// SIMATIC S7-200 project (STEP 7-Micro/WIN), CPU 224 CN REL 02.01

SYMBOL_TABLE 用户定义1
缺料故障             M11.3
急停故障             M11.2
立箱不成功故障          M11.1
折盖回              T99
上升               Q1.0
下降               Q1.1
主机零位脉冲           M4.1
系统运行             M4.0
主机零位接近           I0.1
启动               I1.1
停止               I1.2
复位               I2.5
缺料光电             I2.2
红灯               Q0.2
绿灯               Q0.3
黄灯               Q0.5
主1速              Q0.4
主2速              Q0.6
主3速              Q0.7
吸箱真空             Q2.0
吸箱气缸             Q2.1
抹箱               Q2.3
折盖               Q2.4
固箱               Q2.5
上夹               Q2.6
下放               Q2.7
固箱真空             Q3.1
左推               Q3.2
右推               Q3.3
屏启动              V10.0
屏停止              V10.1
停箱脉冲光电           I2.7
满箱报警             M13.3
满箱光电             I1.0
END_SYMBOL_TABLE

ORGANIZATION_BLOCK 主程序:OB1
TITLE=程序注释
BEGIN
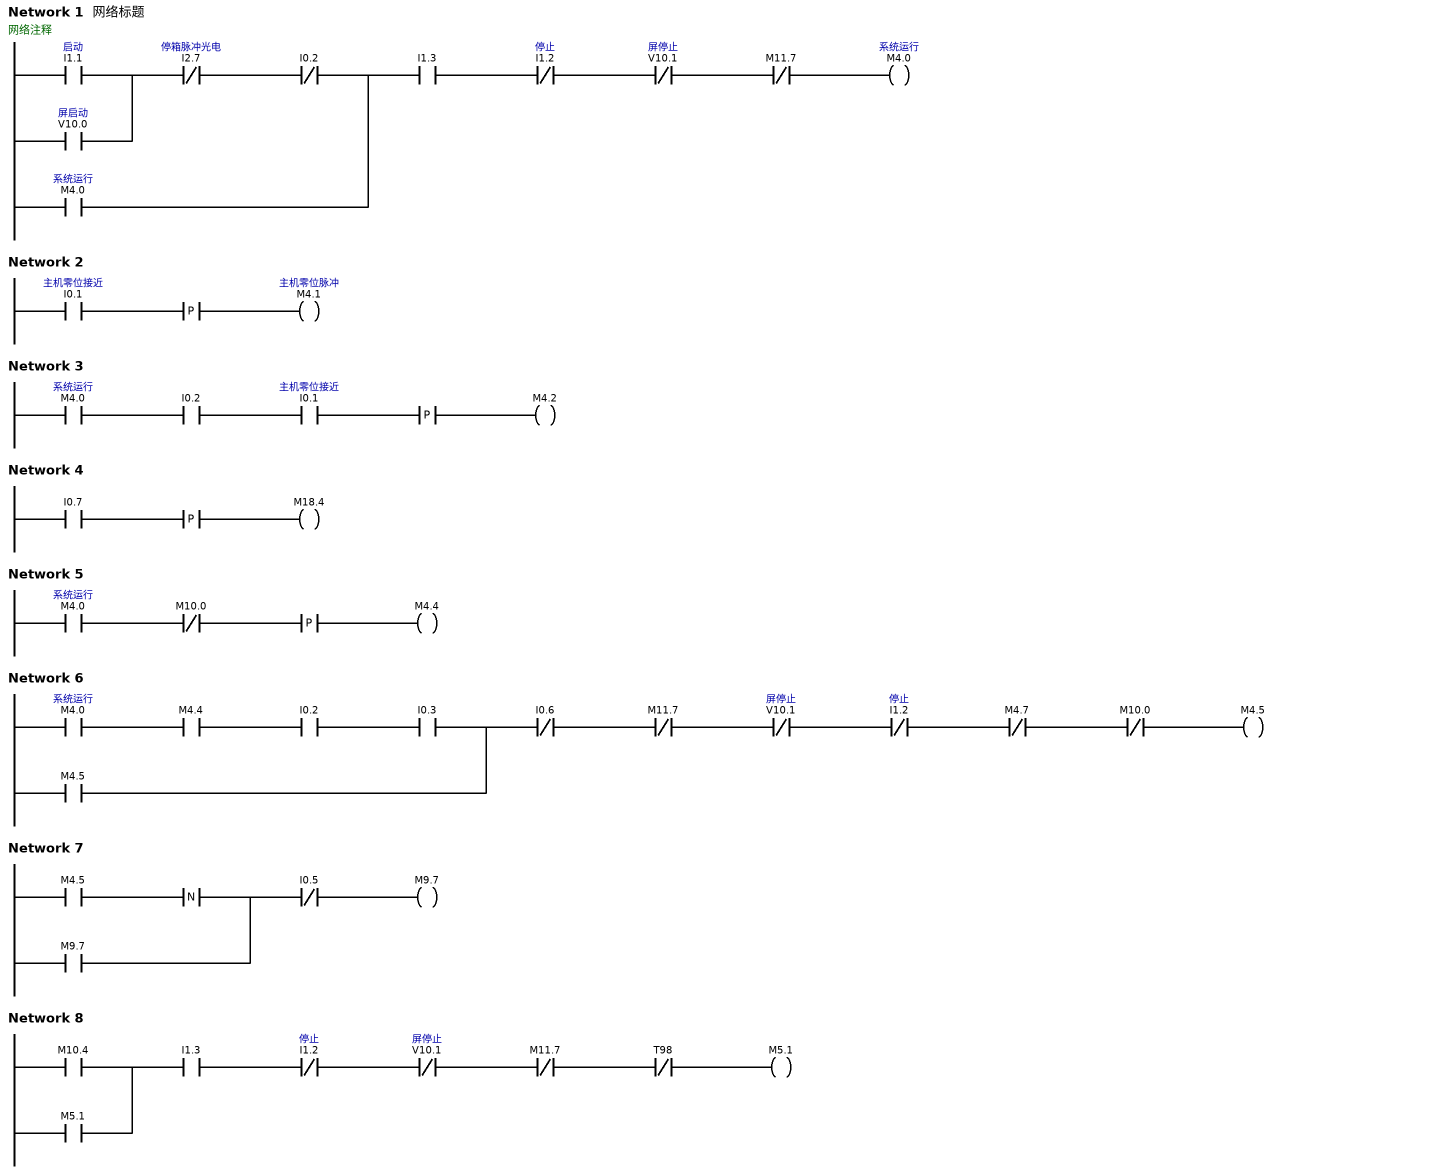
Network 1 // 网络标题
// 网络注释
LD     启动:I1.1
O      屏启动:V10.0
AN     停箱脉冲光电:I2.7
AN     I0.2
O      系统运行:M4.0
A      I1.3
AN     停止:I1.2
AN     屏停止:V10.1
AN     M11.7
=      系统运行:M4.0
Network 2
LD     主机零位接近:I0.1
EU
=      主机零位脉冲:M4.1
Network 3
LD     系统运行:M4.0
A      I0.2
A      主机零位接近:I0.1
EU
=      M4.2
Network 4
LD     I0.7
EU
=      M18.4
Network 5
LD     系统运行:M4.0
AN     M10.0
EU
=      M4.4
Network 6
LD     系统运行:M4.0
A      M4.4
A      I0.2
A      I0.3
O      M4.5
AN     I0.6
AN     M11.7
AN     屏停止:V10.1
AN     停止:I1.2
AN     M4.7
AN     M10.0
=      M4.5
Network 7
LD     M4.5
ED
O      M9.7
AN     I0.5
=      M9.7
Network 8
LD     M10.4
O      M5.1
A      I1.3
AN     停止:I1.2
AN     屏停止:V10.1
AN     M11.7
AN     T98
=      M5.1
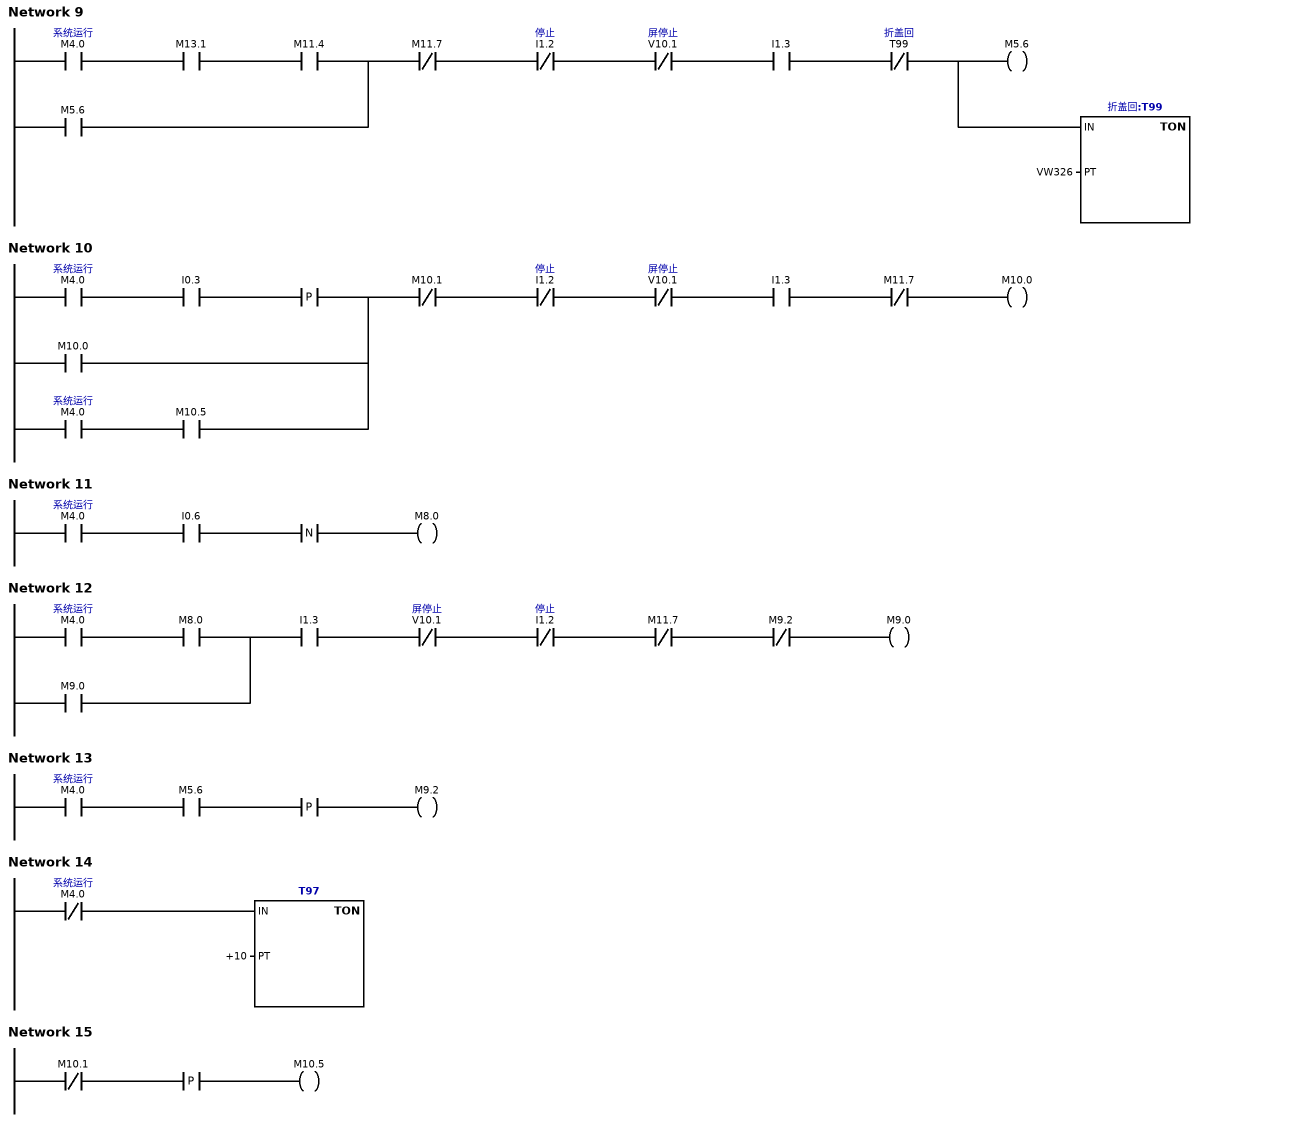
Network 9
LD     系统运行:M4.0
A      M13.1
A      M11.4
O      M5.6
AN     M11.7
AN     停止:I1.2
AN     屏停止:V10.1
A      I1.3
AN     折盖回:T99
=      M5.6
TON    折盖回:T99, VW326
Network 10
LD     系统运行:M4.0
A      I0.3
EU
O      M10.0
LD     系统运行:M4.0
A      M10.5
OLD
AN     M10.1
AN     停止:I1.2
AN     屏停止:V10.1
A      I1.3
AN     M11.7
=      M10.0
Network 11
LD     系统运行:M4.0
A      I0.6
ED
=      M8.0
Network 12
LD     系统运行:M4.0
A      M8.0
O      M9.0
A      I1.3
AN     屏停止:V10.1
AN     停止:I1.2
AN     M11.7
AN     M9.2
=      M9.0
Network 13
LD     系统运行:M4.0
A      M5.6
EU
=      M9.2
Network 14
LDN    系统运行:M4.0
TON    T97, +10
Network 15
LDN    M10.1
EU
=      M10.5
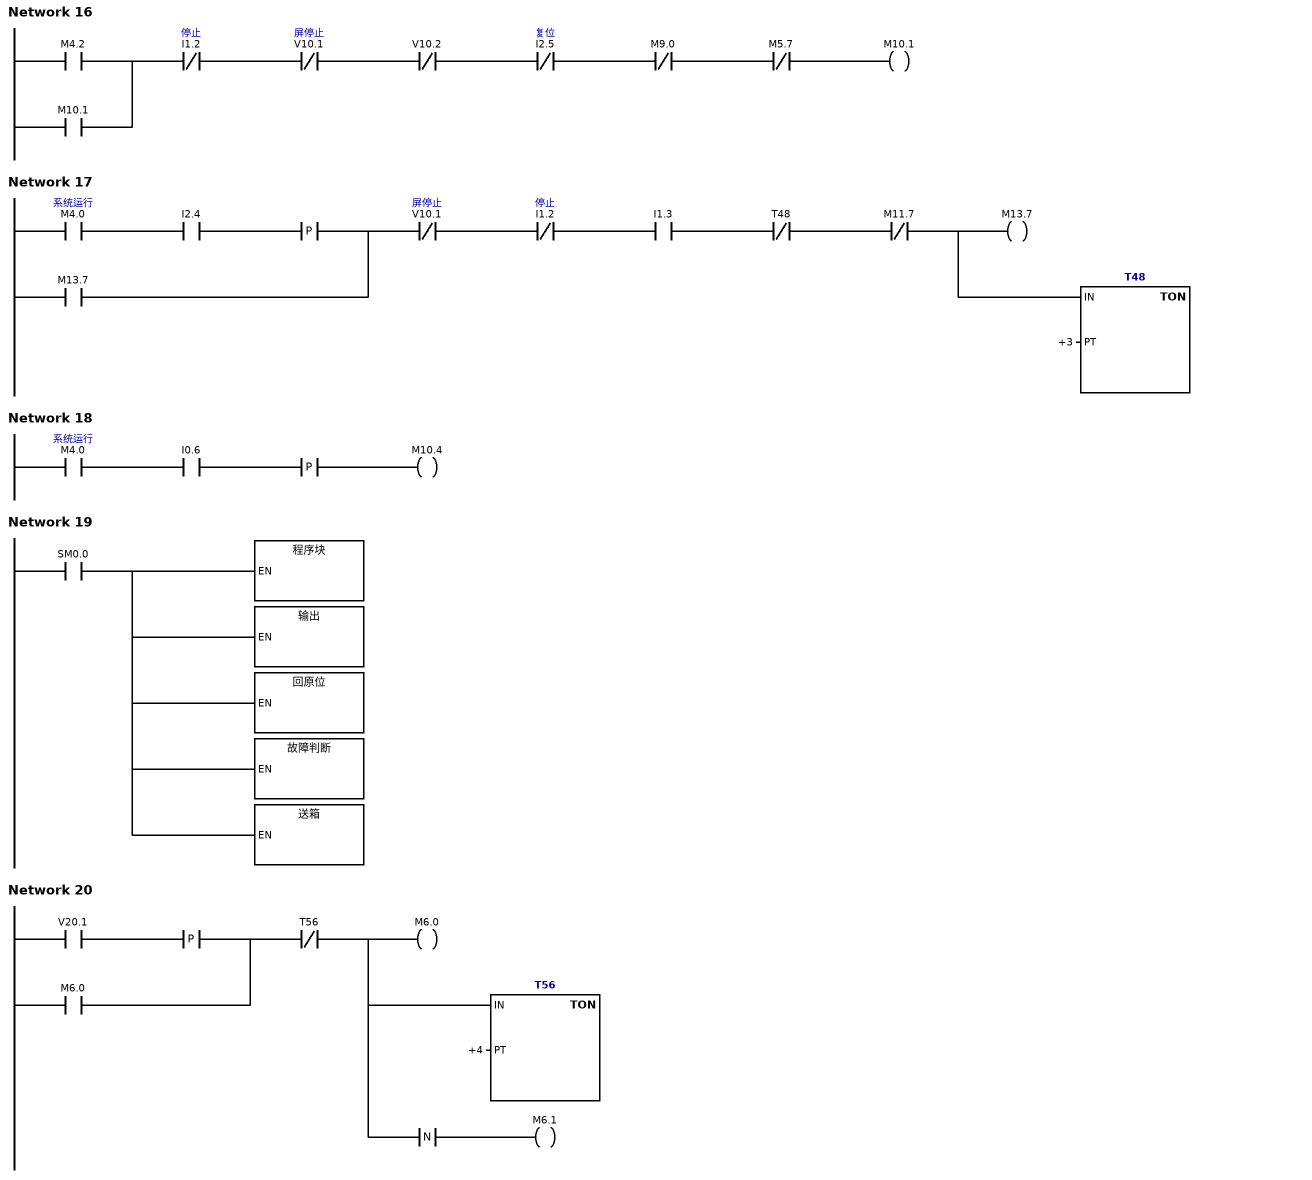
Network 16
LD     M4.2
O      M10.1
AN     停止:I1.2
AN     屏停止:V10.1
AN     V10.2
AN     复位:I2.5
AN     M9.0
AN     M5.7
=      M10.1
Network 17
LD     系统运行:M4.0
A      I2.4
EU
O      M13.7
AN     屏停止:V10.1
AN     停止:I1.2
A      I1.3
AN     T48
AN     M11.7
=      M13.7
TON    T48, +3
Network 18
LD     系统运行:M4.0
A      I0.6
EU
=      M10.4
Network 19
LD     SM0.0
CALL   程序块:SBR0
CALL   输出:SBR1
CALL   回原位:SBR4
CALL   故障判断:SBR3
CALL   送箱:SBR2
Network 20
LD     V20.1
EU
O      M6.0
AN     T56
=      M6.0
TON    T56, +4
ED
=      M6.1
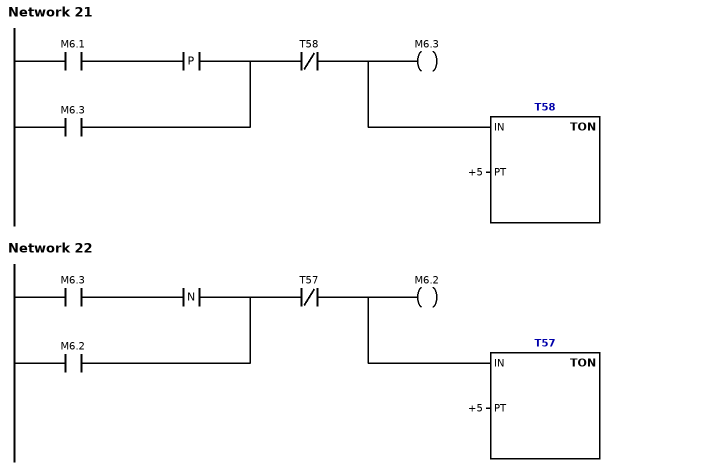
Network 21
LD     M6.1
EU
O      M6.3
AN     T58
=      M6.3
TON    T58, +5
Network 22
LD     M6.3
ED
O      M6.2
AN     T57
=      M6.2
TON    T57, +5
END_ORGANIZATION_BLOCK

SUBROUTINE_BLOCK 程序块:SBR0
TITLE=子程序注释
BEGIN
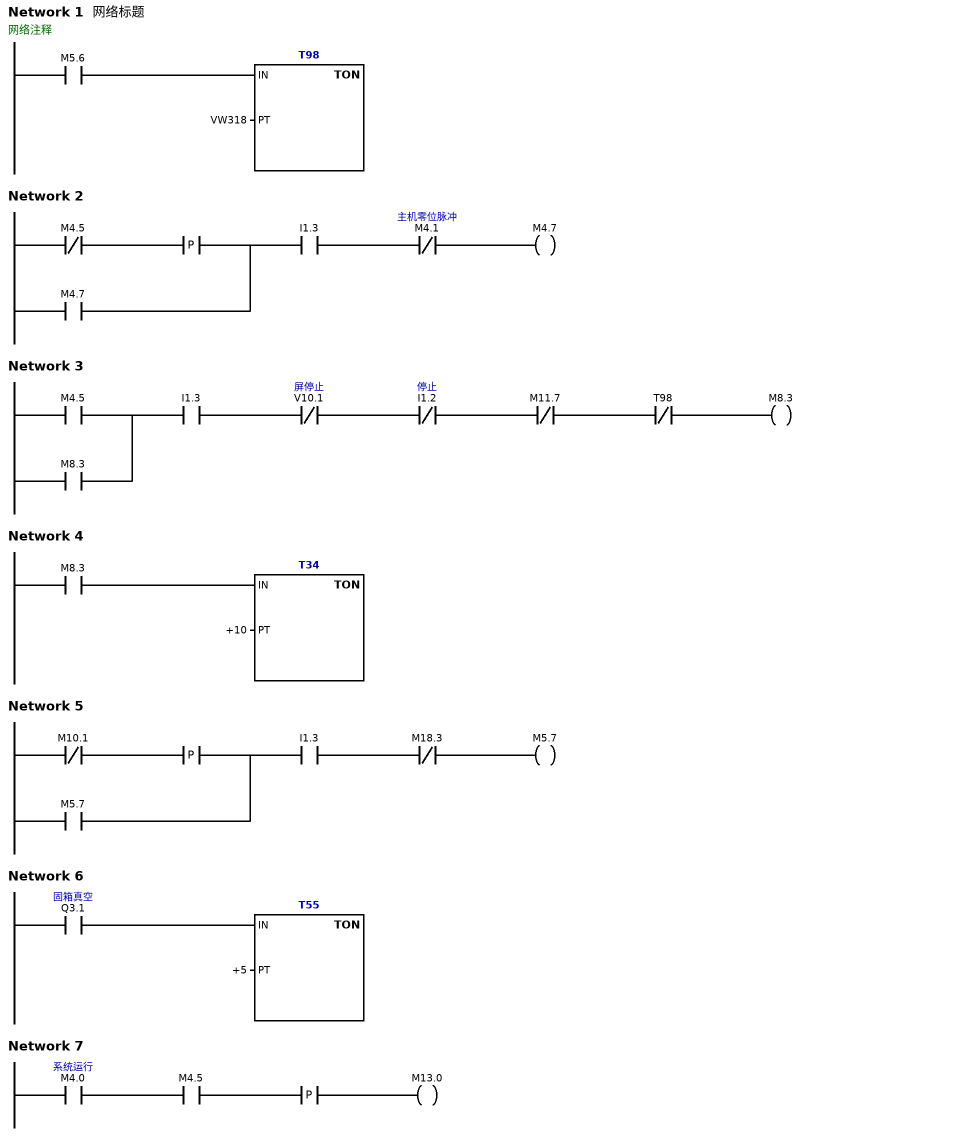
Network 1 // 网络标题
// 网络注释
LD     M5.6
TON    T98, VW318
Network 2
LDN    M4.5
EU
O      M4.7
A      I1.3
AN     主机零位脉冲:M4.1
=      M4.7
Network 3
LD     M4.5
O      M8.3
A      I1.3
AN     屏停止:V10.1
AN     停止:I1.2
AN     M11.7
AN     T98
=      M8.3
Network 4
LD     M8.3
TON    T34, +10
Network 5
LDN    M10.1
EU
O      M5.7
A      I1.3
AN     M18.3
=      M5.7
Network 6
LD     固箱真空:Q3.1
TON    T55, +5
Network 7
LD     系统运行:M4.0
A      M4.5
EU
=      M13.0
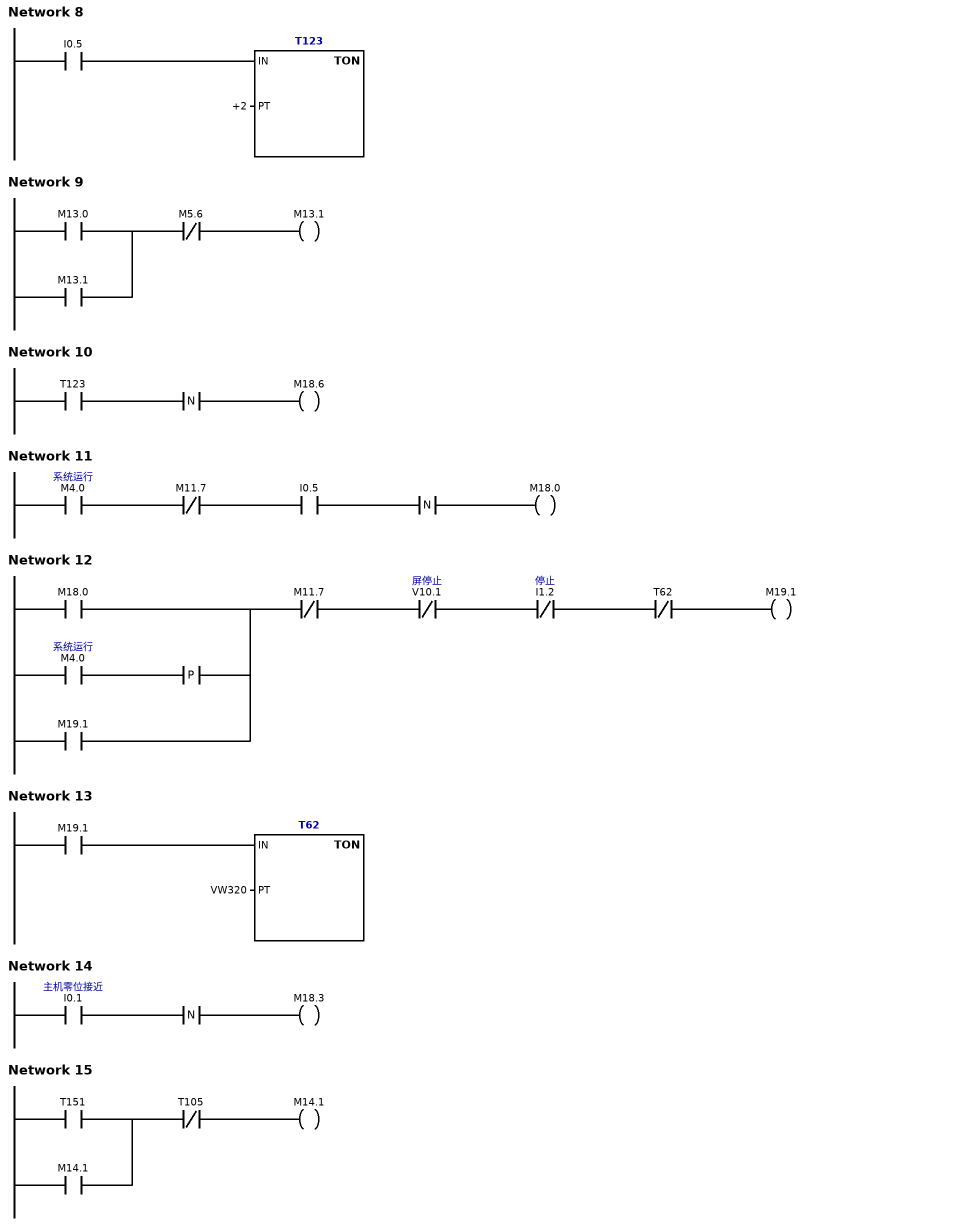
Network 8
LD     I0.5
TON    T123, +2
Network 9
LD     M13.0
O      M13.1
AN     M5.6
=      M13.1
Network 10
LD     T123
ED
=      M18.6
Network 11
LD     系统运行:M4.0
AN     M11.7
A      I0.5
ED
=      M18.0
Network 12
LD     M18.0
LD     系统运行:M4.0
EU
OLD
O      M19.1
AN     M11.7
AN     屏停止:V10.1
AN     停止:I1.2
AN     T62
=      M19.1
Network 13
LD     M19.1
TON    T62, VW320
Network 14
LD     主机零位接近:I0.1
ED
=      M18.3
Network 15
LD     T151
O      M14.1
AN     T105
=      M14.1
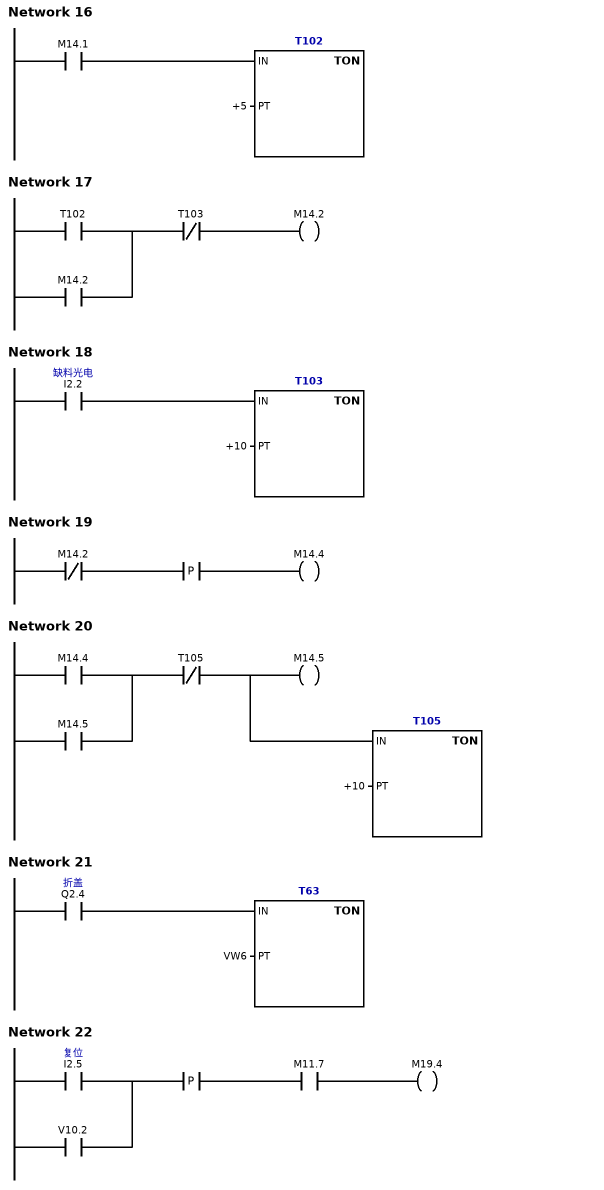
Network 16
LD     M14.1
TON    T102, +5
Network 17
LD     T102
O      M14.2
AN     T103
=      M14.2
Network 18
LD     缺料光电:I2.2
TON    T103, +10
Network 19
LDN    M14.2
EU
=      M14.4
Network 20
LD     M14.4
O      M14.5
AN     T105
=      M14.5
TON    T105, +10
Network 21
LD     折盖:Q2.4
TON    T63, VW6
Network 22
LD     复位:I2.5
O      V10.2
EU
A      M11.7
=      M19.4
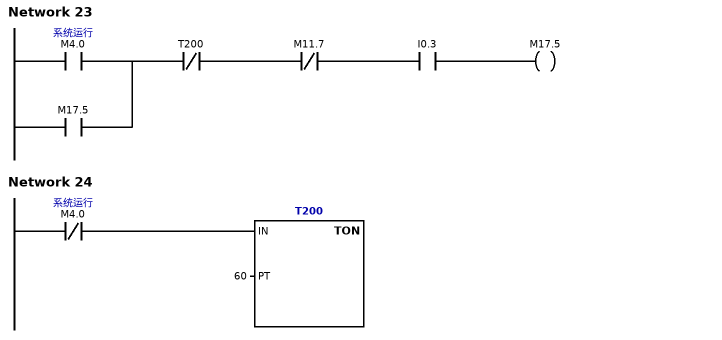
Network 23
LD     系统运行:M4.0
O      M17.5
AN     T200
AN     M11.7
A      I0.3
=      M17.5
Network 24
LDN    系统运行:M4.0
TON    T200, 60
END_SUBROUTINE_BLOCK

SUBROUTINE_BLOCK 输出:SBR1
TITLE=子程序注释
BEGIN
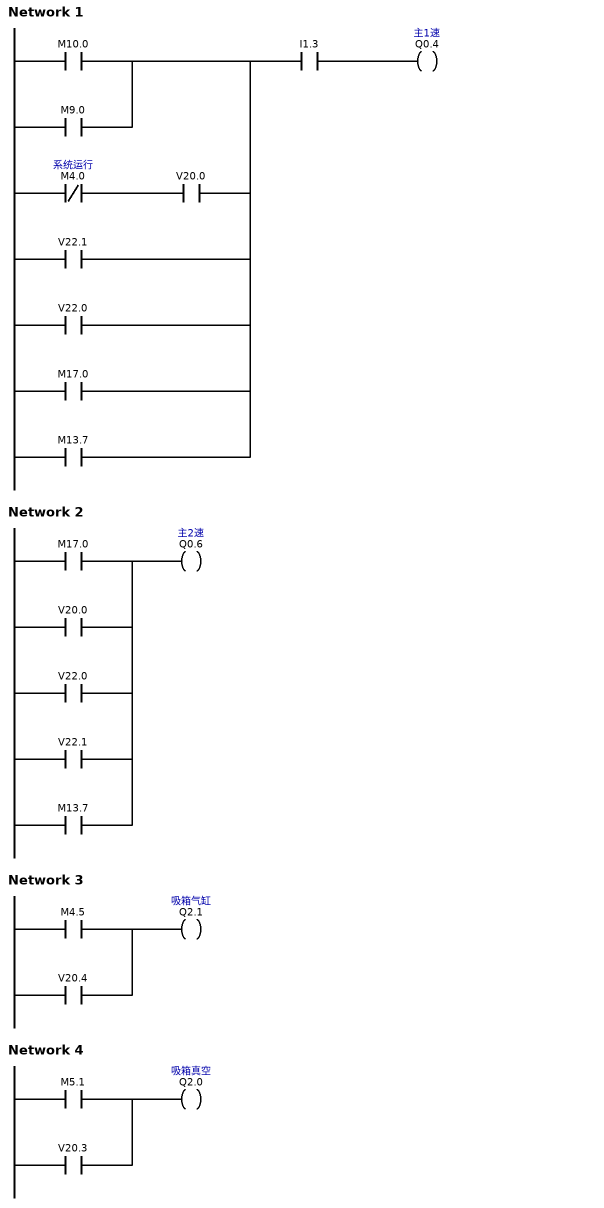
Network 1
LD     M10.0
O      M9.0
LDN    系统运行:M4.0
A      V20.0
OLD
O      V22.1
O      V22.0
O      M17.0
O      M13.7
A      I1.3
=      主1速:Q0.4
Network 2
LD     M17.0
O      V20.0
O      V22.0
O      V22.1
O      M13.7
=      主2速:Q0.6
Network 3
LD     M4.5
O      V20.4
=      吸箱气缸:Q2.1
Network 4
LD     M5.1
O      V20.3
=      吸箱真空:Q2.0
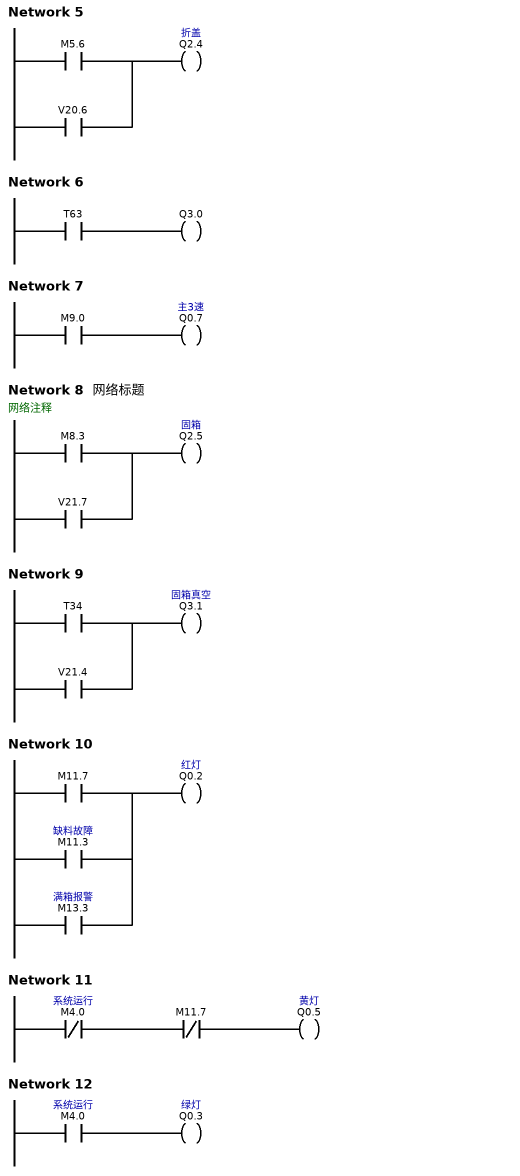
Network 5
LD     M5.6
O      V20.6
=      折盖:Q2.4
Network 6
LD     T63
=      Q3.0
Network 7
LD     M9.0
=      主3速:Q0.7
Network 8 // 网络标题
// 网络注释
LD     M8.3
O      V21.7
=      固箱:Q2.5
Network 9
LD     T34
O      V21.4
=      固箱真空:Q3.1
Network 10
LD     M11.7
O      缺料故障:M11.3
O      满箱报警:M13.3
=      红灯:Q0.2
Network 11
LDN    系统运行:M4.0
AN     M11.7
=      黄灯:Q0.5
Network 12
LD     系统运行:M4.0
=      绿灯:Q0.3
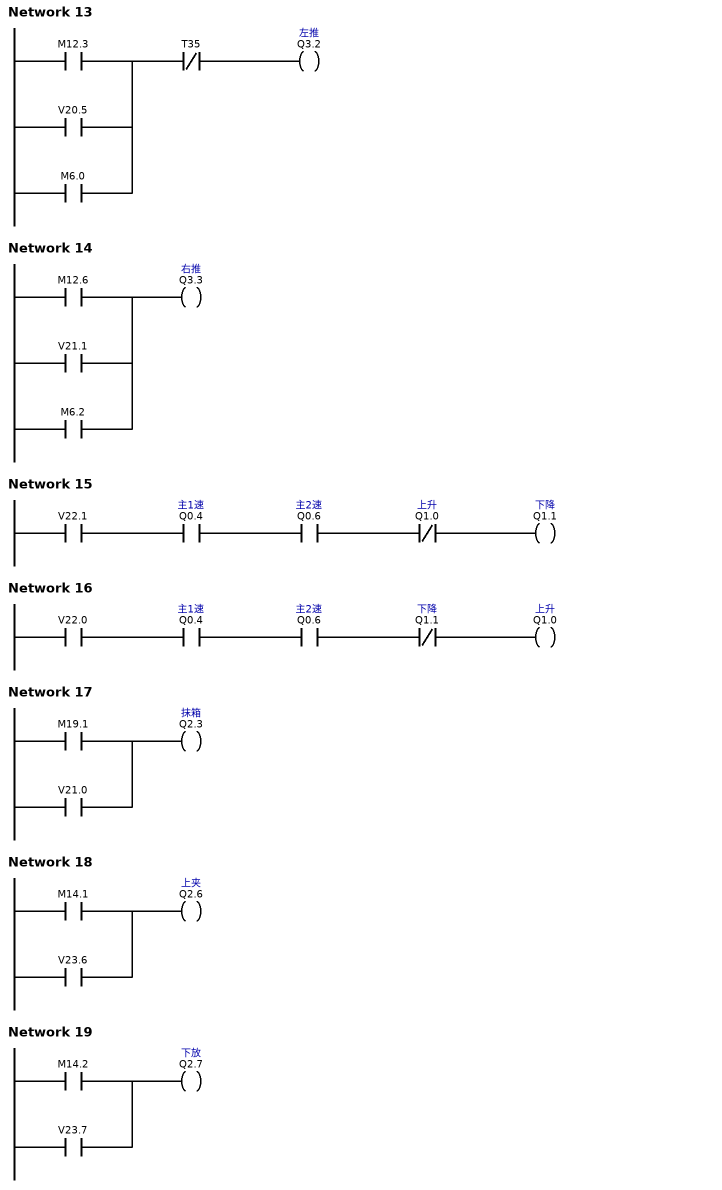
Network 13
LD     M12.3
O      V20.5
O      M6.0
AN     T35
=      左推:Q3.2
Network 14
LD     M12.6
O      V21.1
O      M6.2
=      右推:Q3.3
Network 15
LD     V22.1
A      主1速:Q0.4
A      主2速:Q0.6
AN     上升:Q1.0
=      下降:Q1.1
Network 16
LD     V22.0
A      主1速:Q0.4
A      主2速:Q0.6
AN     下降:Q1.1
=      上升:Q1.0
Network 17
LD     M19.1
O      V21.0
=      抹箱:Q2.3
Network 18
LD     M14.1
O      V23.6
=      上夹:Q2.6
Network 19
LD     M14.2
O      V23.7
=      下放:Q2.7
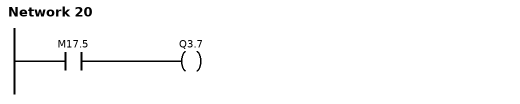
Network 20
LD     M17.5
=      Q3.7
END_SUBROUTINE_BLOCK

SUBROUTINE_BLOCK 送箱:SBR2
TITLE=子程序注释
BEGIN
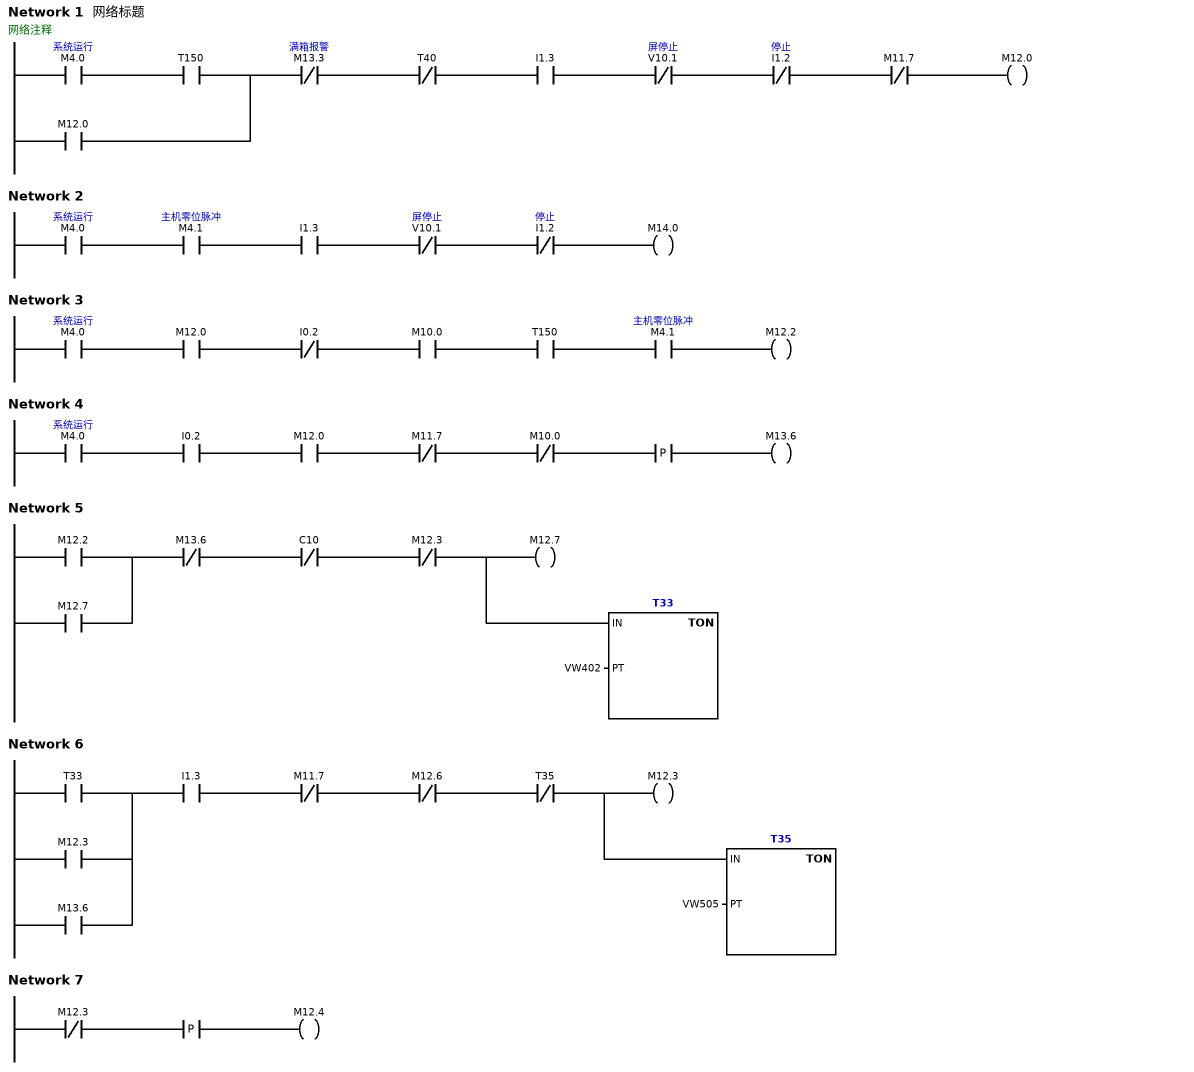
Network 1 // 网络标题
// 网络注释
LD     系统运行:M4.0
A      T150
O      M12.0
AN     满箱报警:M13.3
AN     T40
A      I1.3
AN     屏停止:V10.1
AN     停止:I1.2
AN     M11.7
=      M12.0
Network 2
LD     系统运行:M4.0
A      主机零位脉冲:M4.1
A      I1.3
AN     屏停止:V10.1
AN     停止:I1.2
=      M14.0
Network 3
LD     系统运行:M4.0
A      M12.0
AN     I0.2
A      M10.0
A      T150
A      主机零位脉冲:M4.1
=      M12.2
Network 4
LD     系统运行:M4.0
A      I0.2
A      M12.0
AN     M11.7
AN     M10.0
EU
=      M13.6
Network 5
LD     M12.2
O      M12.7
AN     M13.6
AN     C10
AN     M12.3
=      M12.7
TON    T33, VW402
Network 6
LD     T33
O      M12.3
O      M13.6
A      I1.3
AN     M11.7
AN     M12.6
AN     T35
=      M12.3
TON    T35, VW505
Network 7
LDN    M12.3
EU
=      M12.4
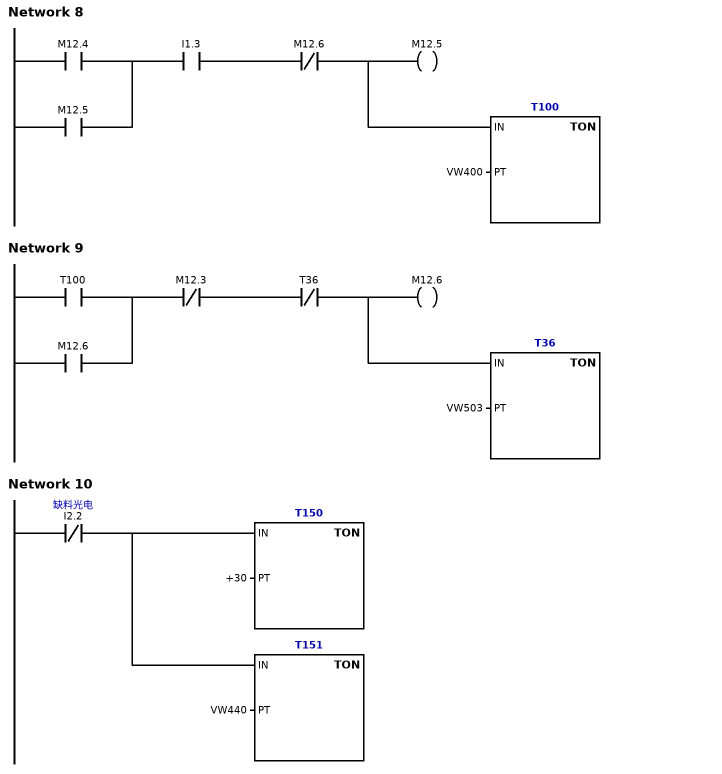
Network 8
LD     M12.4
O      M12.5
A      I1.3
AN     M12.6
=      M12.5
TON    T100, VW400
Network 9
LD     T100
O      M12.6
AN     M12.3
AN     T36
=      M12.6
TON    T36, VW503
Network 10
LDN    缺料光电:I2.2
TON    T150, +30
TON    T151, VW440
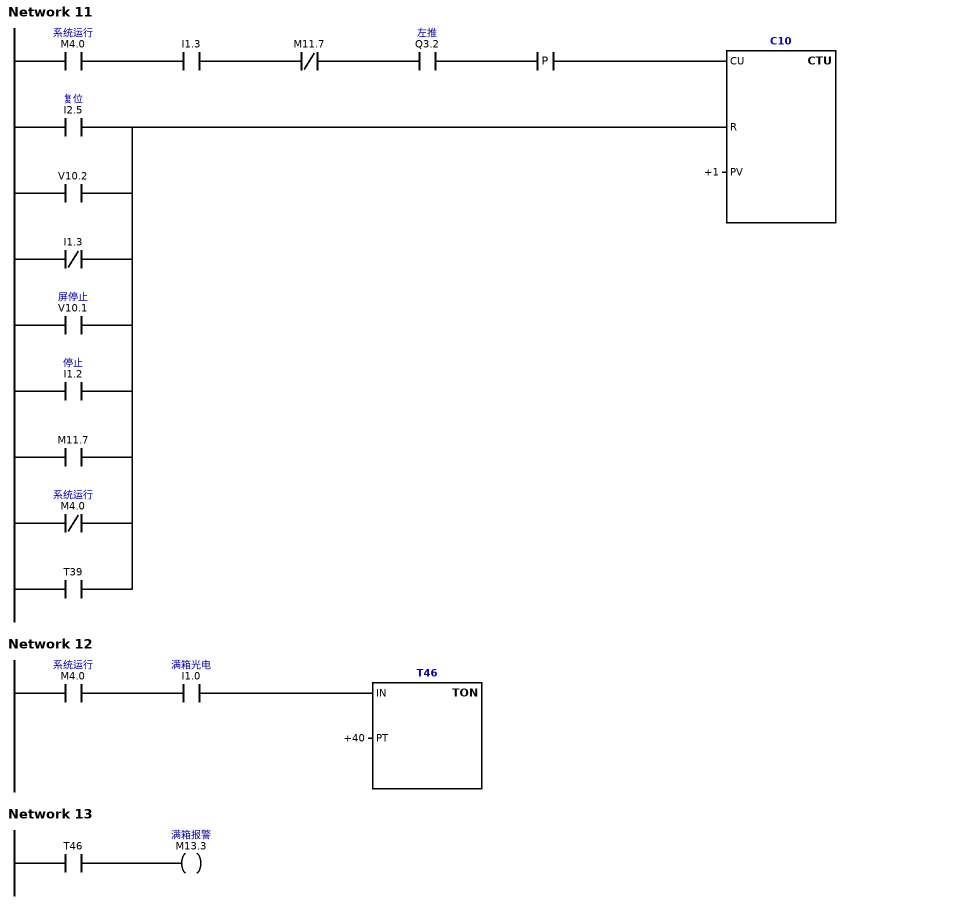
Network 11
LD     系统运行:M4.0
A      I1.3
AN     M11.7
A      左推:Q3.2
EU
LD     复位:I2.5
O      V10.2
ON     I1.3
O      屏停止:V10.1
O      停止:I1.2
O      M11.7
ON     系统运行:M4.0
O      T39
CTU    C10, +1
Network 12
LD     系统运行:M4.0
A      满箱光电:I1.0
TON    T46, +40
Network 13
LD     T46
=      满箱报警:M13.3
END_SUBROUTINE_BLOCK

SUBROUTINE_BLOCK 故障判断:SBR3
TITLE=子程序注释
BEGIN
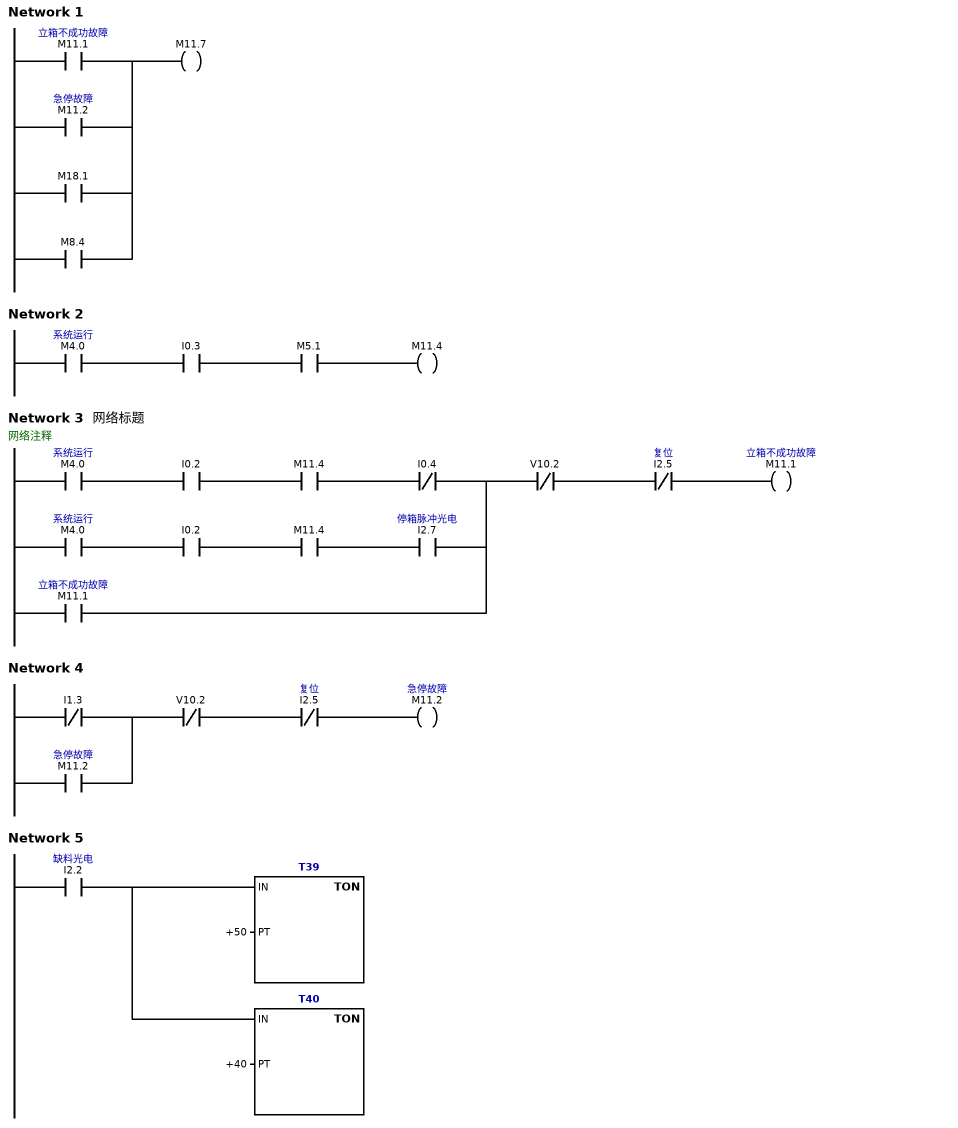
Network 1
LD     立箱不成功故障:M11.1
O      急停故障:M11.2
O      M18.1
O      M8.4
=      M11.7
Network 2
LD     系统运行:M4.0
A      I0.3
A      M5.1
=      M11.4
Network 3 // 网络标题
// 网络注释
LD     系统运行:M4.0
A      I0.2
A      M11.4
AN     I0.4
LD     系统运行:M4.0
A      I0.2
A      M11.4
A      停箱脉冲光电:I2.7
OLD
O      立箱不成功故障:M11.1
AN     V10.2
AN     复位:I2.5
=      立箱不成功故障:M11.1
Network 4
LDN    I1.3
O      急停故障:M11.2
AN     V10.2
AN     复位:I2.5
=      急停故障:M11.2
Network 5
LD     缺料光电:I2.2
TON    T39, +50
TON    T40, +40
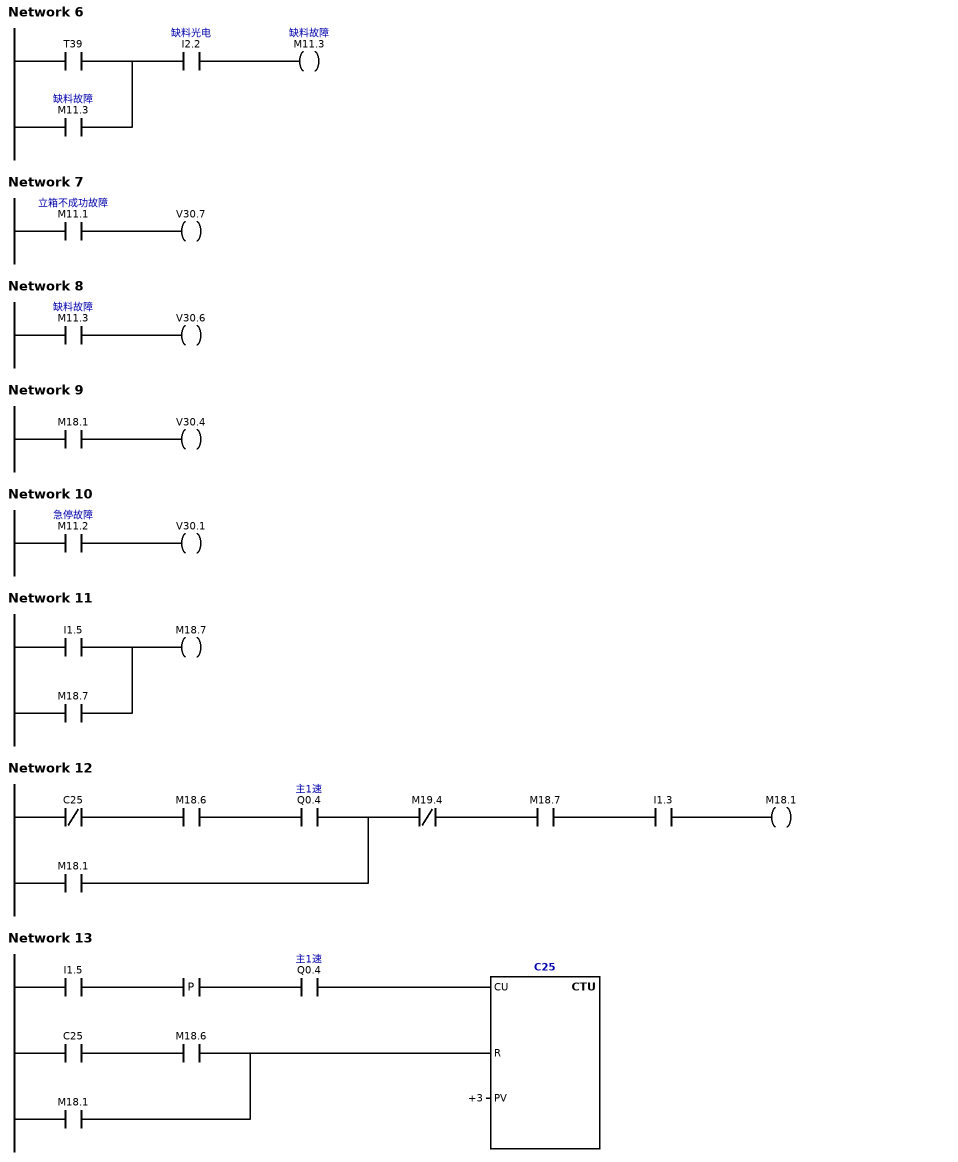
Network 6
LD     T39
O      缺料故障:M11.3
A      缺料光电:I2.2
=      缺料故障:M11.3
Network 7
LD     立箱不成功故障:M11.1
=      V30.7
Network 8
LD     缺料故障:M11.3
=      V30.6
Network 9
LD     M18.1
=      V30.4
Network 10
LD     急停故障:M11.2
=      V30.1
Network 11
LD     I1.5
O      M18.7
=      M18.7
Network 12
LDN    C25
A      M18.6
A      主1速:Q0.4
O      M18.1
AN     M19.4
A      M18.7
A      I1.3
=      M18.1
Network 13
LD     I1.5
EU
A      主1速:Q0.4
LD     C25
A      M18.6
O      M18.1
CTU    C25, +3
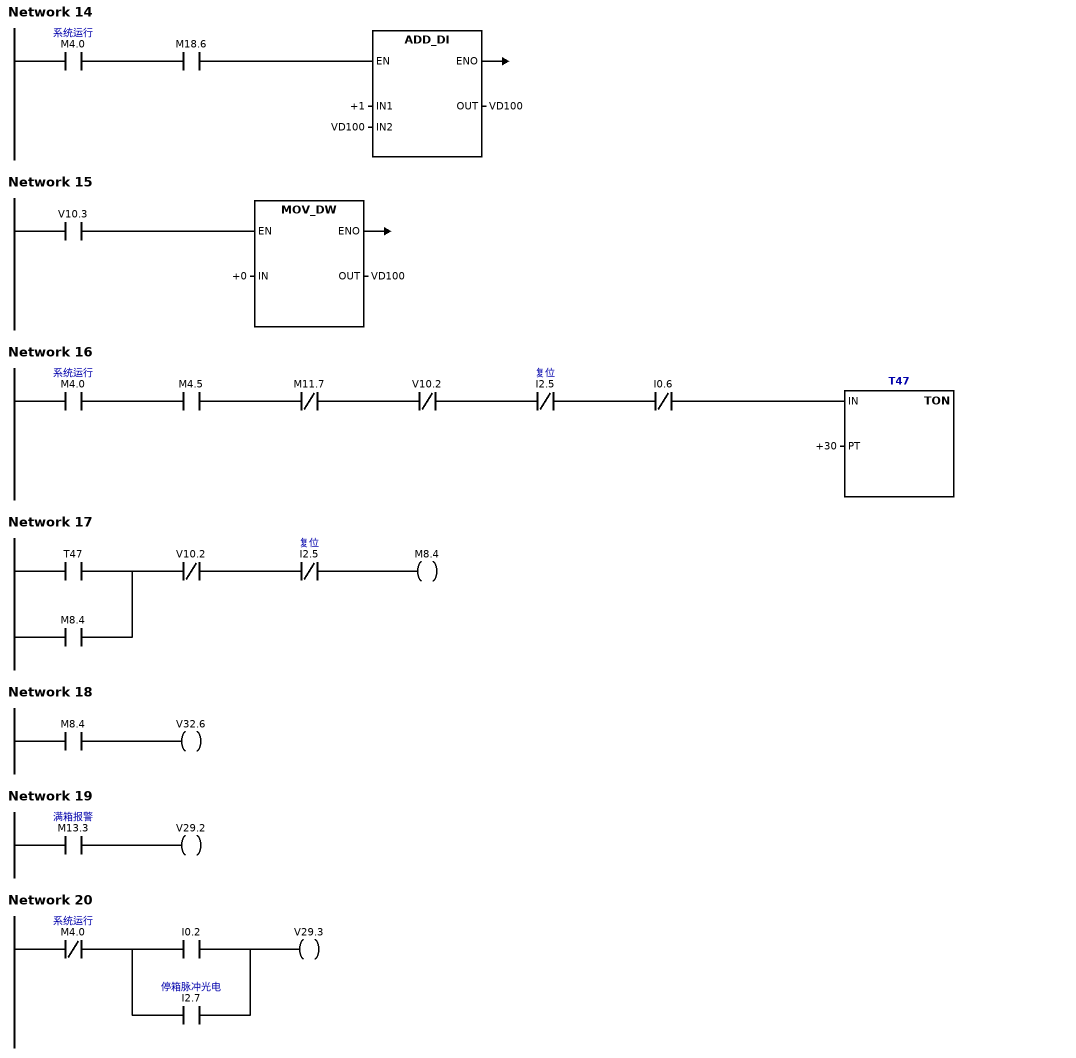
Network 14
LD     系统运行:M4.0
A      M18.6
+D     +1, VD100
Network 15
LD     V10.3
MOVD   +0, VD100
Network 16
LD     系统运行:M4.0
A      M4.5
AN     M11.7
AN     V10.2
AN     复位:I2.5
AN     I0.6
TON    T47, +30
Network 17
LD     T47
O      M8.4
AN     V10.2
AN     复位:I2.5
=      M8.4
Network 18
LD     M8.4
=      V32.6
Network 19
LD     满箱报警:M13.3
=      V29.2
Network 20
LDN    系统运行:M4.0
LD     I0.2
O      停箱脉冲光电:I2.7
ALD
=      V29.3
END_SUBROUTINE_BLOCK

SUBROUTINE_BLOCK 回原位:SBR4
TITLE=子程序注释
BEGIN
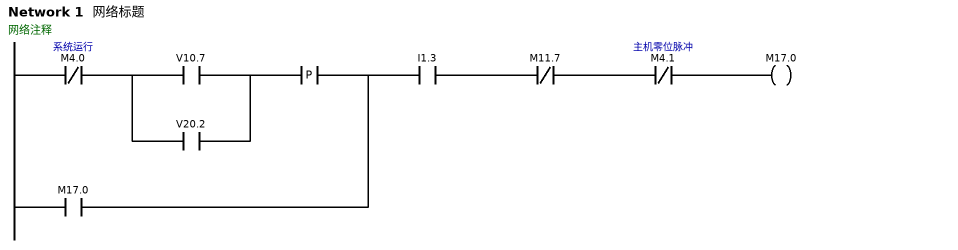
Network 1 // 网络标题
// 网络注释
LDN    系统运行:M4.0
LD     V10.7
O      V20.2
ALD
EU
O      M17.0
A      I1.3
AN     M11.7
AN     主机零位脉冲:M4.1
=      M17.0
END_SUBROUTINE_BLOCK

SUBROUTINE_BLOCK 喷胶:SBR5
TITLE=子程序注释
BEGIN
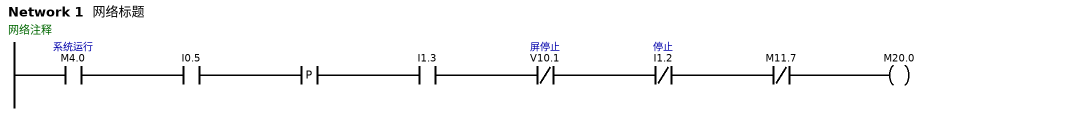
Network 1 // 网络标题
// 网络注释
LD     系统运行:M4.0
A      I0.5
EU
A      I1.3
AN     屏停止:V10.1
AN     停止:I1.2
AN     M11.7
=      M20.0
END_SUBROUTINE_BLOCK
